# EPICS StreamDevice protocol: environmentmonitorSup/environmentmonitor.proto
Terminator = CR;

getTempA {

	out "?STS";
	in "TA%f,RHA%*f,TB%*f,RHB%*f";

}

getTempB {

	out "?STS";
	in "TA%*f,RHA%*f,TB%f,RHB%*f";

}

getRHumidityA {

	out "?STS";
	in "TA%*f,RHA%f,TB%*f,RHB%*f";

}

getRHumidityB {

	out "?STS";
	in "TA%*f,RHA%*f,TB%*f,RHB%f";

}
